// TwinCAT 3 PLC project UnitTests
// Title: Unit Tests for Simple Unit test Lib
// Company: Red Rock Controls Limited
// Author: R Christopher
// ProjectVersion: 1.0.0.0
// ProgramVersion: 3.1.4023.0
// libraries:
//   Tc2_System, * (Beckhoff Automation GmbH)
//   Tc2_Utilities, * (Beckhoff Automation GmbH)
//   Tc3_Module, * (Beckhoff Automation GmbH)
//   tcl_UnitTestLibrary, * (Red Rock Controls Limited)
// project tree:
//   / GlobalTextList.TcGTLO
//   GVLs/ UnitTests.TcGVL
//   POUs/ PB_TestRunner.TcPOU, TestFramework.TcPOU
//   Tasks/ PlcTask.TcTTO
//   Unit Tests/Assertion Tests/ Test_AssertEquals_BLOB_SizeDiffers.TcPOU (excluded from build), Test_AssertEquals_BLOB_TypeClassDiffers.TcPOU (excluded from build), Test_AssertEquals_BLOB_TypeContentDiffers.TcPOU (excluded from build), Test_AssertEquals_BOOL.TcPOU (excluded from build), Test_AssertEquals_BYTE.TcPOU (excluded from build), Test_AssertEquals_DINT.TcPOU (excluded from build), Test_AssertEquals_DWORD.TcPOU (excluded from build), Test_AssertEquals_INT.TcPOU (excluded from build), Test_AssertEquals_INTERFACE.TcPOU (excluded from build), Test_AssertEquals_LINT.TcPOU (excluded from build), Test_AssertEquals_LREAL.TcPOU (excluded from build), Test_AssertEquals_PVOID.TcPOU (excluded from build), Test_AssertEquals_REAL.TcPOU (excluded from build), Test_AssertEquals_STRING.TcPOU (excluded from build), Test_AssertEquals_UDINT.TcPOU (excluded from build), Test_AssertEquals_UINT.TcPOU (excluded from build), Test_AssertEquals_ULINT.TcPOU (excluded from build), Test_AssertEquals_WORD.TcPOU (excluded from build), Test_F_Assert_INTS_Differ.TcPOU
//   Unit Tests/Fixtures/ I_ExampleInterface.TcIO (excluded from build), T_ExampleInterfaceImplementation.TcPOU (excluded from build), T_UnitTestUnderTest.TcPOU (excluded from build)
//   Unit Tests/List Of Tests/ Test_GetTestHandlesInvalidIndex.TcPOU (excluded from build), Test_GetTestReturnsCorrectTest.TcPOU (excluded from build), Test_GetTestHandlesEmptyList.TcPOU (excluded from build), Test_IteratorReturnsTests.TcPOU (excluded from build), Test_ListCountIncrements.TcPOU (excluded from build)
//   Unit Tests/T_UnitTest Tests/ Test_ExampleTest.TcPOU (excluded from build), Test_setTestName_setsTestName.TcPOU (excluded from build)
// (motion and I/O tree: see PLC project tcl_unittestlibrary)
// real-time tasks:
//   TASK PlcTask: cycle T#10ms, priority 20, ADS port 351

CONFIGURATION UnitTests
    RESOURCE PLC ON TwinCAT3
        TASK PlcTask(INTERVAL := T#10ms, PRIORITY := 20);
        PROGRAM PB_TestRunner WITH PlcTask : PB_TestRunner;
    END_RESOURCE
END_CONFIGURATION

// ---- GVLs/UnitTests.TcGVL
{attribute 'qualified_only'}
VAR_GLOBAL
//    TestList : T_ListOfTests(Capacity      := 20,
//                             TestGroupName := 'tcl_UnitTestLibrary');

//	Test_F_Assert_INTS_Differ : Test_F_Assert_INTS_Differ;
						 
//    Test_ListCountIncrements                  : Test_ListCountIncrements(TestList);
//    Test_GetTestReturnsCorrectTest            : Test_GetTestReturnsCorrectTest(TestList);
//    Test_GetTestHandlesEmptyList              : Test_GetTestHandlesEmptyList(TestList);
//    Test_GetTestHandlesInvalidIndex           : Test_GetTestHandlesInvalidIndex(TestList);
//    Test_IteratorReturnsTests                 : Test_IteratorReturnsTests(TestList);
//    Test_ExampleTest                          : Test_ExampleTest(TestList);
//    Test_setTestName_setsTestName             : Test_setTestName_setsTestName(TestList);
//    Test_AssertEquals_BOOL                    : Test_AssertEquals_BOOL(TestList);
//    Test_AssertEquals_BYTE                    : Test_AssertEquals_BYTE(TestList);
//    Test_AssertEquals_DINT                    : Test_AssertEquals_DINT(TestList);
//    Test_AssertEquals_INT                     : Test_AssertEquals_INT(TestList);
//    Test_AssertEquals_INTERFACE               : Test_AssertEquals_INTERFACE(TestList);
//    Test_AssertEquals_LINT                    : Test_AssertEquals_LINT(TestList);
//    Test_AssertEquals_LREAL                   : Test_AssertEquals_LREAL(TestList);
//    Test_AssertEquals_PVOID                   : Test_AssertEquals_PVOID(TestList);
//    Test_AssertEquals_REAL                    : Test_AssertEquals_REAL(TestList);
//    Test_AssertEquals_STRING                  : Test_AssertEquals_STRING(TestList);
//    Test_AssertEquals_UDINT                   : Test_AssertEquals_UDINT(TestList);
//    Test_AssertEquals_UINT                    : Test_AssertEquals_UINT(TestList);
//    Test_AssertEquals_ULINT                   : Test_AssertEquals_ULINT(TestList);
//    Test_AssertEquals_WORD                    : Test_AssertEquals_WORD(TestList);
//    Test_AssertEquals_DWORD                   : Test_AssertEquals_DWORD(TestList);
//    Test_AssertEquals_BLOB_SizeDiffers        : Test_AssertEquals_BLOB_SizeDiffers(TestList);
//    Test_AssertEquals_BLOB_TypeClassDiffers   : Test_AssertEquals_BLOB_TypeClassDiffers(TestList);
//    Test_AssertEquals_BLOB_TypeContentDiffers : Test_AssertEquals_BLOB_TypeContentDiffers(TestList);

//    TestRunner : T_TestRunner(TestList := UnitTests.TestList,
//                              Verbose  := FALSE);
END_VAR

// ---- Unit Tests/Fixtures/I_ExampleInterface.TcIO
INTERFACE I_ExampleInterface EXTENDS __SYSTEM.IQueryInterface

END_INTERFACE

// ---- POUs/PB_TestRunner.TcPOU
PROGRAM PB_TestRunner
VAR
TestFramework : TestFramework;
END_VAR

TestFramework();

//UnitTests.TestRunner();

END_PROGRAM

// ---- POUs/TestFramework.TcPOU
FUNCTION_BLOCK TestFramework
VAR
    Test_F_Assert_INTS_Differ : Test_F_Assert_INTS_Differ;

    //    Test_ListCountIncrements                  : Test_ListCountIncrements(TestList);
    //    Test_GetTestReturnsCorrectTest            : Test_GetTestReturnsCorrectTest(TestList);
    //    Test_GetTestHandlesEmptyList              : Test_GetTestHandlesEmptyList(TestList);
    //    Test_GetTestHandlesInvalidIndex           : Test_GetTestHandlesInvalidIndex(TestList);
    //    Test_IteratorReturnsTests                 : Test_IteratorReturnsTests(TestList);
    //    Test_ExampleTest                          : Test_ExampleTest(TestList);
    //    Test_setTestName_setsTestName             : Test_setTestName_setsTestName(TestList);
    //    Test_AssertEquals_BOOL                    : Test_AssertEquals_BOOL(TestList);
    //    Test_AssertEquals_BYTE                    : Test_AssertEquals_BYTE(TestList);
    //    Test_AssertEquals_DINT                    : Test_AssertEquals_DINT(TestList);
    //    Test_AssertEquals_INT                     : Test_AssertEquals_INT(TestList);
    //    Test_AssertEquals_INTERFACE               : Test_AssertEquals_INTERFACE(TestList);
    //    Test_AssertEquals_LINT                    : Test_AssertEquals_LINT(TestList);
    //    Test_AssertEquals_LREAL                   : Test_AssertEquals_LREAL(TestList);
    //    Test_AssertEquals_PVOID                   : Test_AssertEquals_PVOID(TestList);
    //    Test_AssertEquals_REAL                    : Test_AssertEquals_REAL(TestList);
    //    Test_AssertEquals_STRING                  : Test_AssertEquals_STRING(TestList);
    //    Test_AssertEquals_UDINT                   : Test_AssertEquals_UDINT(TestList);
    //    Test_AssertEquals_UINT                    : Test_AssertEquals_UINT(TestList);
    //    Test_AssertEquals_ULINT                   : Test_AssertEquals_ULINT(TestList);
    //    Test_AssertEquals_WORD                    : Test_AssertEquals_WORD(TestList);
    //    Test_AssertEquals_DWORD                   : Test_AssertEquals_DWORD(TestList);
    //    Test_AssertEquals_BLOB_SizeDiffers        : Test_AssertEquals_BLOB_SizeDiffers(TestList);
    //    Test_AssertEquals_BLOB_TypeClassDiffers   : Test_AssertEquals_BLOB_TypeClassDiffers(TestList);
    //    Test_AssertEquals_BLOB_TypeContentDiffers : Test_AssertEquals_BLOB_TypeContentDiffers(TestList);

    TestRunner              : T_TestRunner;
    OnlineChangeCount       : UDINT;
    StoredOnlineChangeCount : UDINT := 100;
END_VAR

OnlineChangeCount := TwinCAT_SystemInfoVarList._AppInfo.OnlineChangeCnt;
IF OnlineChangeCount <> StoredOnlineChangeCount THEN
    StoredOnlineChangeCount := OnlineChangeCount;

    TestRunner.Init();
    TestRunner.AddTest(Test_F_Assert_INTS_Differ);
    TestRunner.Start();
END_IF

TestRunner();

END_FUNCTION_BLOCK

// ---- Unit Tests/Assertion Tests/Test_F_Assert_INTS_Differ.TcPOU
FUNCTION_BLOCK Test_F_Assert_INTS_Differ EXTENDS T_UnitTestBase

METHOD  Init : BOOL
State := 0;
END_METHOD

METHOD RunTest
VAR_OUTPUT
    TestCompleted : BOOL;
    TestFailed    : BOOL;
END_VAR
VAR
    AssertionResult : BOOL;
    Expected        : INT;
    Actual          : INT;
END_VAR
Expected := 133;
Actual   := 133;

AssertionResult := F_Assert(Source       := THIS^.TestName,
                            Expected     := Expected,
                            Actual       := Actual,
                            VariableName := 'F_Assert()');

IF AssertionResult = FALSE THEN
    TestFailed := TRUE;
END_IF
TestCompleted := TRUE;
END_METHOD

END_FUNCTION_BLOCK

// ---- Unit Tests/List Of Tests/Test_ListCountIncrements.TcPOU
FUNCTION_BLOCK Test_ListCountIncrements EXTENDS T_UnitTestBase
VAR
    List  : T_ListOfTests(Capacity := 10, TestGroupName := 'Unit Tests');
    Test1 : T_UnitTestBase(List);
END_VAR

Assertion.AssertEquals_DINT(Expected     := 1,
                            Actual       := List.Count,
                            VariableName := 'List.Count');
							
CheckAssertion(NextState := 0);

END_FUNCTION_BLOCK

// ---- Unit Tests/List Of Tests/Test_GetTestReturnsCorrectTest.TcPOU
FUNCTION_BLOCK Test_GetTestReturnsCorrectTest EXTENDS T_UnitTestBase
VAR
	List : T_ListOfTests(Capacity := 10,TestGroupName := 'Unit Tests');
	Test1 : T_UnitTestBase(List);
	Test2 : T_UnitTestBase(List);
	Test3 : T_UnitTestBase(List);
	Test4 : T_UnitTestBase(List);
	
	Result : I_UnitTest;
END_VAR

Result := List.GetTest(2);


Assertion.AssertEquals_STRING(Expected     := 'Test3',
                            Actual       := Result.TestName,
                            VariableName := 'Result.TestName');
							
CheckAssertion(NextState := 0);

END_FUNCTION_BLOCK

// ---- Unit Tests/List Of Tests/Test_GetTestHandlesEmptyList.TcPOU
FUNCTION_BLOCK Test_GetTestHandlesEmptyList EXTENDS T_UnitTestBase
VAR
	List : T_ListOfTests(Capacity := 10,TestGroupName := 'Unit Tests');
	Result : I_UnitTest;
END_VAR

List.Clear();

Result := List.GetTest(2);

Assertion.AssertEquals_INTERFACE(Expected     := 0,
                            Actual       := Result,
                            VariableName := 'GetTest()');
							
CheckAssertion(NextState := 0);

END_FUNCTION_BLOCK

// ---- Unit Tests/List Of Tests/Test_GetTestHandlesInvalidIndex.TcPOU
FUNCTION_BLOCK Test_GetTestHandlesInvalidIndex EXTENDS T_UnitTestBase
VAR
    List   : T_ListOfTests(Capacity := 10,TestGroupName := 'Unit Tests');
    Test1  : T_UnitTestBase(List);
    Test2  : T_UnitTestBase(List);
    Test3  : T_UnitTestBase(List);
    Test4  : T_UnitTestBase(List);
    Result : I_UnitTest;
END_VAR

Result := List.GetTest(4);

Assertion.AssertEquals_INTERFACE(Expected     := 0,
                                 Actual       := Result,
                                 VariableName := 'GetTest()');

CheckAssertion(NextState := 0);

END_FUNCTION_BLOCK

// ---- Unit Tests/List Of Tests/Test_IteratorReturnsTests.TcPOU
FUNCTION_BLOCK Test_IteratorReturnsTests EXTENDS T_UnitTestBase
VAR
    List     : T_ListOfTests(Capacity := 10,TestGroupName := 'Unit Tests');
    Iterator : T_TestIterator;
    Test1    : T_UnitTestBase(List);
    Test2    : T_UnitTestBase(List);
    Test3    : T_UnitTestBase(List);
    Test4    : T_UnitTestBase(List);

    Result : I_UnitTest;
END_VAR

Iterator.Initialise(List);
Iterator.GetNext();
Iterator.GetNext();
Result := Iterator.GetNext();

Assertion.AssertEquals_STRING(Expected     := 'Test3',
                              Actual       := Result.TestName,
                              VariableName := 'List.Count');

CheckAssertion(NextState := 0);

END_FUNCTION_BLOCK

// ---- Unit Tests/T_UnitTest Tests/Test_ExampleTest.TcPOU
FUNCTION_BLOCK Test_ExampleTest EXTENDS T_UnitTestBase IMPLEMENTS I_UnitTest
VAR_INPUT
END_VAR
VAR_OUTPUT
END_VAR
VAR
	TestByte : BYTE := 123;
END_VAR

Assertion.AssertEquals_BYTE(Expected     := 123,
                            Actual       := TestByte,
                            VariableName := 'TestByte');

CheckAssertion(NextState := 0);

END_FUNCTION_BLOCK

// ---- Unit Tests/T_UnitTest Tests/Test_setTestName_setsTestName.TcPOU
FUNCTION_BLOCK Test_setTestName_setsTestName EXTENDS T_UnitTestBase
VAR_INPUT
END_VAR
VAR_OUTPUT
END_VAR
VAR
    List     : T_ListOfTests(Capacity := 10, TestGroupName := 'Unit Tests');
    UnitTest : T_UnitTestUnderTest(List);
END_VAR

UnitTest.setTestName();

Assertion.AssertEquals_STRING(Expected     := 'UnitTest',
                              Actual       := UnitTest._TestName,
                              VariableName := 'UnitTest.TestName');

CheckAssertion(NextState := 0);

END_FUNCTION_BLOCK

// ---- Unit Tests/Fixtures/T_UnitTestUnderTest.TcPOU
FUNCTION_BLOCK T_UnitTestUnderTest EXTENDS T_UnitTestBase
VAR_INPUT
END_VAR
VAR_OUTPUT
END_VAR
VAR
END_VAR

END_FUNCTION_BLOCK

// ---- Unit Tests/Assertion Tests/Test_AssertEquals_BOOL.TcPOU
FUNCTION_BLOCK Test_AssertEquals_BOOL EXTENDS T_UnitTestBase
VAR
    AssertionUnderTest : T_Assertion;
    BOOL_Variable : BOOL := FALSE;
END_VAR

// Test the assertion...
AssertionUnderTest.AssertEquals_BOOL(
    Expected := TRUE,
    Actual   := BOOL_Variable,
    VariableName := 'BOOL_Variable');
    
// Assert that the assertion failed...
Assertion.AssertEquals_BOOL(Expected     := TRUE,
                            Actual       := AssertionUnderTest.AssertionFailed,
                            VariableName := 'AssertionUnderTest.AssertionFailed');

// Check the assertion worked...  
CheckAssertion(NextState := 0);

END_FUNCTION_BLOCK

// ---- Unit Tests/Assertion Tests/Test_AssertEquals_BYTE.TcPOU
FUNCTION_BLOCK Test_AssertEquals_BYTE EXTENDS T_UnitTestBase
VAR
    AssertionUnderTest : T_Assertion;
    BYTE_Variable : BYTE := 123;
END_VAR


// Test the assertion...
AssertionUnderTest.AssertEquals_BYTE(
    Expected := 234,
    Actual   := BYTE_Variable,
    VariableName := 'BYTE_Variable');
 
// Assert that the assertion failed...
Assertion.AssertEquals_BOOL(Expected     := TRUE,
                            Actual       := AssertionUnderTest.AssertionFailed,
                            VariableName := 'AssertionUnderTest.AssertionFailed');

// Check the assertion worked...  
CheckAssertion(NextState := 0);

END_FUNCTION_BLOCK

// ---- Unit Tests/Assertion Tests/Test_AssertEquals_DINT.TcPOU
FUNCTION_BLOCK Test_AssertEquals_DINT EXTENDS T_UnitTestBase
VAR
    AssertionUnderTest : T_Assertion;
    DINT_Variable : DINT := 1111;
END_VAR

// Test the assertion...
AssertionUnderTest.AssertEquals_DINT(
    Expected := 2222,
    Actual   := DINT_Variable,
    VariableName := 'DINT_Variable');
    
// Assert that the assertion failed...
Assertion.AssertEquals_BOOL(Expected     := TRUE,
                            Actual       := AssertionUnderTest.AssertionFailed,
                            VariableName := 'AssertionUnderTest.AssertionFailed');

// Check the assertion worked...  
CheckAssertion(NextState := 0);

END_FUNCTION_BLOCK

// ---- Unit Tests/Assertion Tests/Test_AssertEquals_INT.TcPOU
FUNCTION_BLOCK Test_AssertEquals_INT EXTENDS T_UnitTestBase
VAR
    AssertionUnderTest : T_Assertion;
    INT_Variable : INT := 1111;
END_VAR

// Test the assertion...
AssertionUnderTest.AssertEquals_INT(
    Expected := 2222,
    Actual   := INT_Variable,
    VariableName := 'INT_Variable');
 
// Assert that the assertion failed...
Assertion.AssertEquals_BOOL(Expected     := TRUE,
                            Actual       := AssertionUnderTest.AssertionFailed,
                            VariableName := 'AssertionUnderTest.AssertionFailed');

// Check the assertion worked...  
CheckAssertion(NextState := 0);

END_FUNCTION_BLOCK

// ---- Unit Tests/Assertion Tests/Test_AssertEquals_INTERFACE.TcPOU
FUNCTION_BLOCK Test_AssertEquals_INTERFACE EXTENDS T_UnitTestBase
VAR
    AssertionUnderTest : T_Assertion;
    
    ExampleInterfaceImplementation1   : T_ExampleInterfaceImplementation;
    INTERFACE_Variable1 : I_ExampleInterface := ExampleInterfaceImplementation1;
    
    ExampleInterfaceImplementation2   : T_ExampleInterfaceImplementation;
    INTERFACE_Variable2 : I_ExampleInterface := ExampleInterfaceImplementation2;
END_VAR

// Test the assertion...
AssertionUnderTest.AssertEquals_INTERFACE(
    Expected := INTERFACE_Variable1,
    Actual   := INTERFACE_Variable2,
    VariableName := 'INTERFACE_Variable2'); 
    
// Assert that the assertion failed...
Assertion.AssertEquals_BOOL(Expected     := TRUE,
                            Actual       := AssertionUnderTest.AssertionFailed,
                            VariableName := 'AssertionUnderTest.AssertionFailed');

// Check the assertion worked...  
CheckAssertion(NextState := 0);

END_FUNCTION_BLOCK

// ---- Unit Tests/Fixtures/T_ExampleInterfaceImplementation.TcPOU
FUNCTION_BLOCK T_ExampleInterfaceImplementation IMPLEMENTS I_ExampleInterface
VAR_INPUT
END_VAR
VAR_OUTPUT
END_VAR
VAR
END_VAR

END_FUNCTION_BLOCK

// ---- Unit Tests/Assertion Tests/Test_AssertEquals_LINT.TcPOU
FUNCTION_BLOCK Test_AssertEquals_LINT EXTENDS T_UnitTestBase
VAR
    AssertionUnderTest : T_Assertion;
    LINT_Variable : LINT := 1111;
END_VAR

// Test the assertion...
AssertionUnderTest.AssertEquals_LINT(
    Expected := 2222,
    Actual   := LINT_Variable,
    VariableName := 'LINT_Variable');
 
    
// Assert that the assertion failed...
Assertion.AssertEquals_BOOL(Expected     := TRUE,
                            Actual       := AssertionUnderTest.AssertionFailed,
                            VariableName := 'AssertionUnderTest.AssertionFailed');

// Check the assertion worked...  
CheckAssertion(NextState := 0);

END_FUNCTION_BLOCK

// ---- Unit Tests/Assertion Tests/Test_AssertEquals_LREAL.TcPOU
FUNCTION_BLOCK Test_AssertEquals_LREAL EXTENDS T_UnitTestBase
VAR
    AssertionUnderTest : T_Assertion;
    LREAL_Variable : LREAL := 1.111;
END_VAR

// Test the assertion...
AssertionUnderTest.AssertEquals_LREAL(
    Expected := 2.222,
    Actual   := LREAL_Variable,
    Delta    := 0.001,
    VariableName := 'LREAL_Variable');
   
// Assert that the assertion failed...
Assertion.AssertEquals_BOOL(Expected     := TRUE,
                            Actual       := AssertionUnderTest.AssertionFailed,
                            VariableName := 'AssertionUnderTest.AssertionFailed');

// Check the assertion worked...  
CheckAssertion(NextState := 0);

END_FUNCTION_BLOCK

// ---- Unit Tests/Assertion Tests/Test_AssertEquals_PVOID.TcPOU
FUNCTION_BLOCK Test_AssertEquals_PVOID EXTENDS T_UnitTestBase
VAR
    AssertionUnderTest : T_Assertion;
    PVOID_Variable : PVOID := 1111;
END_VAR

// Test the assertion...
AssertionUnderTest.AssertEquals_PVOID(
    Expected := 2222,
    Actual   := PVOID_Variable,
    VariableName := 'PVOID_Variable'); 
    
// Assert that the assertion failed...
Assertion.AssertEquals_BOOL(Expected     := TRUE,
                            Actual       := AssertionUnderTest.AssertionFailed,
                            VariableName := 'AssertionUnderTest.AssertionFailed');

// Check the assertion worked...  
CheckAssertion(NextState := 0);

END_FUNCTION_BLOCK

// ---- Unit Tests/Assertion Tests/Test_AssertEquals_REAL.TcPOU
FUNCTION_BLOCK Test_AssertEquals_REAL EXTENDS T_UnitTestBase
VAR
    AssertionUnderTest : T_Assertion;
    REAL_Variable : REAL := 1.111;
END_VAR

// Test the assertion...
AssertionUnderTest.AssertEquals_REAL(
    Expected := 2.222,
    Actual   := REAL_Variable,
    Delta    := 0.001,
    VariableName := 'REAL_Variable');
  
// Assert that the assertion failed...
Assertion.AssertEquals_BOOL(Expected     := TRUE,
                            Actual       := AssertionUnderTest.AssertionFailed,
                            VariableName := 'AssertionUnderTest.AssertionFailed');

// Check the assertion worked...  
CheckAssertion(NextState := 0);

END_FUNCTION_BLOCK

// ---- Unit Tests/Assertion Tests/Test_AssertEquals_STRING.TcPOU
FUNCTION_BLOCK Test_AssertEquals_STRING EXTENDS T_UnitTestBase
VAR
    AssertionUnderTest : T_Assertion;
    STRING_Variable : STRING := 'Cucumber';
END_VAR

// Test the assertion...
AssertionUnderTest.AssertEquals_STRING(
    Expected := 'Radish',
    Actual   := STRING_Variable,
    VariableName := 'STRING_Variable'); 
    
// Assert that the assertion failed...
Assertion.AssertEquals_BOOL(Expected     := TRUE,
                            Actual       := AssertionUnderTest.AssertionFailed,
                            VariableName := 'AssertionUnderTest.AssertionFailed');

// Check the assertion worked...  
CheckAssertion(NextState := 0);

END_FUNCTION_BLOCK

// ---- Unit Tests/Assertion Tests/Test_AssertEquals_UDINT.TcPOU
FUNCTION_BLOCK Test_AssertEquals_UDINT EXTENDS T_UnitTestBase
VAR
    AssertionUnderTest : T_Assertion;
    UDINT_Variable : UDINT := 1111;
END_VAR

// Test the assertion...
AssertionUnderTest.AssertEquals_UDINT(
    Expected := 2222,
    Actual   := UDINT_Variable,
    VariableName := 'UDINT_Variable');
    
// Assert that the assertion failed...
Assertion.AssertEquals_BOOL(Expected     := TRUE,
                            Actual       := AssertionUnderTest.AssertionFailed,
                            VariableName := 'AssertionUnderTest.AssertionFailed');

// Check the assertion worked...  
CheckAssertion(NextState := 0);

END_FUNCTION_BLOCK

// ---- Unit Tests/Assertion Tests/Test_AssertEquals_UINT.TcPOU
FUNCTION_BLOCK Test_AssertEquals_UINT EXTENDS T_UnitTestBase
VAR
    AssertionUnderTest : T_Assertion;
    UINT_Variable : UINT := 1111;
END_VAR

// Test the assertion...
AssertionUnderTest.AssertEquals_UINT(
    Expected := 2222,
    Actual   := UINT_Variable,
    VariableName := 'UINT_Variable');
   
// Assert that the assertion failed...
Assertion.AssertEquals_BOOL(Expected     := TRUE,
                            Actual       := AssertionUnderTest.AssertionFailed,
                            VariableName := 'AssertionUnderTest.AssertionFailed');

// Check the assertion worked...  
CheckAssertion(NextState := 0);

END_FUNCTION_BLOCK

// ---- Unit Tests/Assertion Tests/Test_AssertEquals_ULINT.TcPOU
FUNCTION_BLOCK Test_AssertEquals_ULINT EXTENDS T_UnitTestBase
VAR
    AssertionUnderTest : T_Assertion;
    ULINT_Variable : ULINT := 1111;
END_VAR

// Test the assertion...
AssertionUnderTest.AssertEquals_ULINT(
    Expected := 2222,
    Actual   := ULINT_Variable,
    VariableName := 'ULINT_Variable');
   
// Assert that the assertion failed...
Assertion.AssertEquals_BOOL(Expected     := TRUE,
                            Actual       := AssertionUnderTest.AssertionFailed,
                            VariableName := 'AssertionUnderTest.AssertionFailed');

// Check the assertion worked...  
CheckAssertion(NextState := 0);

END_FUNCTION_BLOCK

// ---- Unit Tests/Assertion Tests/Test_AssertEquals_WORD.TcPOU
FUNCTION_BLOCK Test_AssertEquals_WORD EXTENDS T_UnitTestBase
VAR
    AssertionUnderTest : T_Assertion;
    WORD_Variable : WORD := 1111;
END_VAR

// Test the assertion...
AssertionUnderTest.AssertEquals_WORD(
    Expected := 2222, // deliberately different to test the assertion
    Actual   := WORD_Variable,
    VariableName := 'WORD_Variable');
 
// Assert that the assertion failed...
Assertion.AssertEquals_BOOL(Expected     := TRUE,
                            Actual       := AssertionUnderTest.AssertionFailed,
                            VariableName := 'AssertionUnderTest.AssertionFailed');

// Check the assertion worked...  
CheckAssertion(NextState := 0);

END_FUNCTION_BLOCK

// ---- Unit Tests/Assertion Tests/Test_AssertEquals_DWORD.TcPOU
FUNCTION_BLOCK Test_AssertEquals_DWORD EXTENDS T_UnitTestBase
VAR
    AssertionUnderTest : T_Assertion;
    DWORD_Variable : DWORD := 1111;
END_VAR

// Test the assertion...
AssertionUnderTest.AssertEquals_DWORD(
    Expected := 2222, // deliberately different to test the assertion
    Actual   := DWORD_Variable,
    VariableName := 'DWORD_Variable');
 
    
// Assert that the assertion failed...
Assertion.AssertEquals_BOOL(Expected     := TRUE,
                            Actual       := AssertionUnderTest.AssertionFailed,
                            VariableName := 'AssertionUnderTest.AssertionFailed');

// Check the assertion worked...  
CheckAssertion(NextState := 0);

END_FUNCTION_BLOCK

// ---- Unit Tests/Assertion Tests/Test_AssertEquals_BLOB_SizeDiffers.TcPOU
FUNCTION_BLOCK Test_AssertEquals_BLOB_SizeDiffers EXTENDS T_UnitTestBase
VAR
    AssertionUnderTest : T_Assertion;
    BYTE_Variable : BYTE := 123;
    WORD_Variable : WORD := 456;
END_VAR

// Test the assertion...
AssertionUnderTest.AssertEquals_BLOB(Expected     := BYTE_Variable,
                                     Actual       := WORD_Variable,
                                     VariableName := 'WORD_Variable');

// Assert that the assertion failed...
Assertion.AssertEquals_BOOL(Expected     := TRUE,
                            Actual       := AssertionUnderTest.AssertionFailed,
                            VariableName := 'AssertionUnderTest.AssertionFailed');

// Check the assertion worked...  
CheckAssertion(NextState := 0);

END_FUNCTION_BLOCK

// ---- Unit Tests/Assertion Tests/Test_AssertEquals_BLOB_TypeClassDiffers.TcPOU
FUNCTION_BLOCK Test_AssertEquals_BLOB_TypeClassDiffers EXTENDS T_UnitTestBase
VAR
    AssertionUnderTest : T_Assertion;
    
    // Sizes are the same, but TypeClass differs...
    INT_Variable  : INT  := 123;
    WORD_Variable : WORD := 123;
END_VAR


// Test the assertion...
AssertionUnderTest.AssertEquals_BLOB(
    Expected := INT_Variable,
    Actual   := WORD_Variable,
    VariableName := 'WORD_Variable');
 
// Assert that the assertion failed...
Assertion.AssertEquals_BOOL(Expected     := TRUE,
                            Actual       := AssertionUnderTest.AssertionFailed,
                            VariableName := 'AssertionUnderTest.AssertionFailed');

// Check the assertion worked...  
CheckAssertion(NextState := 0);

END_FUNCTION_BLOCK

// ---- Unit Tests/Assertion Tests/Test_AssertEquals_BLOB_TypeContentDiffers.TcPOU
FUNCTION_BLOCK Test_AssertEquals_BLOB_TypeContentDiffers EXTENDS T_UnitTestBase
VAR
    AssertionUnderTest : T_Assertion;
    
    // Sizes are the same, but contents differ...
    INT_Variable  : WORD := 123;
    WORD_Variable : WORD := 124;
END_VAR


// Test the assertion...
AssertionUnderTest.AssertEquals_BLOB(
    Expected := INT_Variable,
    Actual   := WORD_Variable,
    VariableName := 'WORD_Variable');
 
// Assert that the assertion failed...
Assertion.AssertEquals_BOOL(Expected     := TRUE,
                            Actual       := AssertionUnderTest.AssertionFailed,
                            VariableName := 'AssertionUnderTest.AssertionFailed');

// Check the assertion worked...  
CheckAssertion(NextState := 0);

END_FUNCTION_BLOCK

// ---- GlobalTextList.TcGTLO
TEXTLIST GlobalTextList
  199 = ' %s'
  708 = 'Abort'
  792 = 'Abort Tests'
  346 = 'Checkbox'
  478 = 'Reload Tests'
  906 = 'Run'
  643 = 'Run Sequentially'
  480 = 'Run Tests'
END_TEXTLIST
